// TIA Portal V18 export
DATA_BLOCK "AHUUnitStates"   // DB103
{ S7_Optimized_Access := 'FALSE' }
VERSION : 0.1
// stored: AutoNumber false, DBAccessibleFromOPCUA true, IsOnlyStoredInLoadMemory false, IsWriteProtectedInAS false
   VAR RETAIN
      UnitStates { S7_SetPoint := 'True'} : "UDT_AHUsState";
   END_VAR
BEGIN
   UnitStates.cPreviousOne[1..2] := 0;
END_DATA_BLOCK
